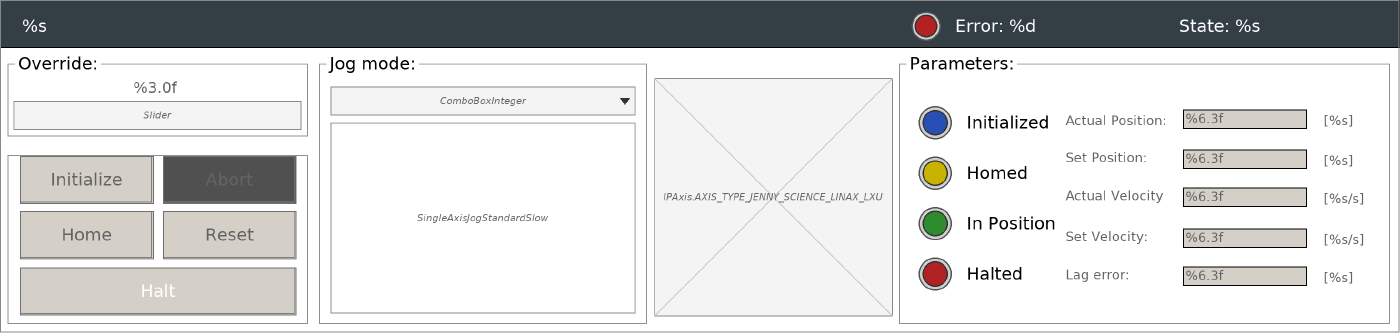
VISUALIZATION SingleAxis_1  // 1470x350
VAR_IN_OUT
	stAxis : ST_VisuCtrlAxisFrame;
END_VAR
    Rectangle (0,0 1470x50)
    Textfield (20,10 699x35), "%s", text variable: stAxis.sName
    Textfield (1235,10 225x35), "State: %s", text list: 'TL_SingleAxisState', text index: stAxis.eAxisState
    Lamp1 (955,10 35x35), variable: stAxis.bError, style: Lamp-Lamp1-Red
    Textfield (1000,10 200x35), "Error: %d", text variable: stAxis.iErrorID
    Image (687,82 250x250), image: IPAxis.AXIS_TYPE_JENNY_SCIENCE_LINAX_LXU
        p84334746: stAxis.sAxisImage
    GroupBox (8,59 315x84), "Override:"
        Slider (6,47 302x30), variable: stAxis.lrOverride, scale 0..100
        Rectangle (55,18 200x30), "%3.0f", text variable: stAxis.lrOverride
    GroupBox (8,155 315x185)
        Button (13,9 140x50), "Initialize"
            tap stAxis.btnInit
        Button (163,9 140x50), "Abort"
            tap stAxis.btnAbort
        Button (13,67 140x50), "Home"
            tap stAxis.btnHome
        Button (163,67 140x50), "Reset"
            tap stAxis.btnReset
        Button (13,126 290x50), "Halt"
            tap stAxis.btnHalt
    GroupBox (335,59 344x281), "Jog mode:"
        Frame (12,70 320x200), frame switch variable: stAxis.eJogMode
            shows SingleAxisJogStandardSlow(btnJogPositive := stAxis.btnJogPositive, btnJogNegative := stAxis.btnJogNegative)
            shows SingleAxisJogStandardFlast(btnJogPositive := stAxis.btnJogPositive, btnJogNegative := stAxis.btnJogNegative)
            shows SingleAxisJogContinous(btnJogPositive := stAxis.btnJogPositive, btnJogNegative := stAxis.btnJogNegative, lrVelocity := stAxis.lrJogVelocity, lrAcceleration := stAxis.lrJogAcceleration, lrDeceleration := stAxis.lrJogDeceleartion, sUnit := stAxis.sUnit)
            shows SingleAxisJogInching(btnJogPositive := stAxis.btnJogPositive, btnJogNegative := stAxis.btnJogNegative, lrPosition := stAxis.lrJogDistance, lrVelocity := stAxis.lrJogVelocity, lrAcceleration := stAxis.lrJogAcceleration, lrDeceleration := stAxis.lrJogDeceleartion, sUnit := stAxis.sUnit)
            shows SingleAxisJogInchingModulo(btnJogPositive := stAxis.btnJogPositive, btnJogNegative := stAxis.btnJogNegative, lrPosition := stAxis.lrJogDistance, lrVelocity := stAxis.lrJogVelocity, lrAcceleration := stAxis.lrJogAcceleration, lrDeceleration := stAxis.lrJogDeceleartion, sUnit := stAxis.sUnit)
        ComboBoxInteger (12,32 320x30), variable: stAxis.eJogMode, text list: 'TL_SingleAxisJogMode'
            p1601986498: ''
    GroupBox (944,59 515x281), "Parameters:"
        Rectangle (298,56 130x20), "%6.3f", text variable: stAxis.lrActualPosition
        Rectangle (443,59 62x18), "[%s]", text variable: stAxis.sUnit
        Rectangle (172,58 110x20), "Actual Position:"
        Lamp1 (18,156 40x40), variable: stAxis.bInPosition, style: Lamp-Lamp1-Green
        Lamp1 (18,50 40x40), variable: stAxis.bActive, style: Lamp-Lamp1-Blue
        Lamp1 (18,103 40x40), variable: stAxis.bHomed, style: Lamp-Lamp1-Yellow
        Label (68,55 100x30), "Initialized"
        Label (68,108 100x30), "Homed"
        Label (68,161 100x30), "In Position"
        Label (68,214 100x30), "Halted"
        Lamp1 (18,209 40x40), variable: stAxis.bHalted, style: Lamp-Lamp1-Red
        Rectangle (172,97 110x20), "Set Position:"
        Rectangle (298,98 130x20), "%6.3f", text variable: stAxis.lrSetPosition
        Rectangle (443,101 62x18), "[%s]", text variable: stAxis.sUnit
        Rectangle (172,137 110x20), "Actual Velocity"
        Rectangle (298,138 130x20), "%6.3f", text variable: stAxis.lrActualVelocity
        Rectangle (443,141 62x18), "[%s/s]", text variable: stAxis.sUnit
        Rectangle (172,180 110x20), "Set Velocity:"
        Rectangle (298,181 130x20), "%6.3f", text variable: stAxis.lrSetVelocity
        Rectangle (443,184 62x18), "[%s/s]", text variable: stAxis.sUnit
        Rectangle (172,220 110x20), "Lag error:"
        Rectangle (298,221 130x20), "%6.3f", text variable: stAxis.lrLagError
        Rectangle (443,224 62x18), "[%s]", text variable: stAxis.sUnit
END_VISUALIZATION

(* stored: Version 1.1.0.1, ProductVersion 3.1.4024.12
   Visu SingleAxis_1: Id {9da82c27-45c5-4a3e-88d8-7f2a125ec19d} *)
